(* Logix 5000 project; controller Sucrose_Main Emulate 5570 rev 20.12; software revision 20.01; part 4 of 30 *)
(* tags used below, declared in another part *)
   AI_E23_0 : REAL[8];   // Analog Input EN2T_FLX 192.168.1.23
   CIPRemote : Area_Program;
   SucroseCIP_PAUSED : BOOL;
   SucroseCIP_RECEIVING_LINE_REMOTE : CIP_REMOTE;
   SucroseCIP_RECEIVING_REMOTE : CIP_REMOTE;
   SucroseCIP_RINGMAIN_REMOTE : CIP_REMOTE;
   SucroseCIP_RUNNING : BOOL;
   SucroseCIP_SeatLift_Pulsing : BOOL;
   SucroseCIP_TK230101_REMOTE : CIP_REMOTE;
(* CIP_RemoteArea_AutoLogic, continued *)

ROUTINE CIP_Receiving_Line_Remote   (* ladder *)
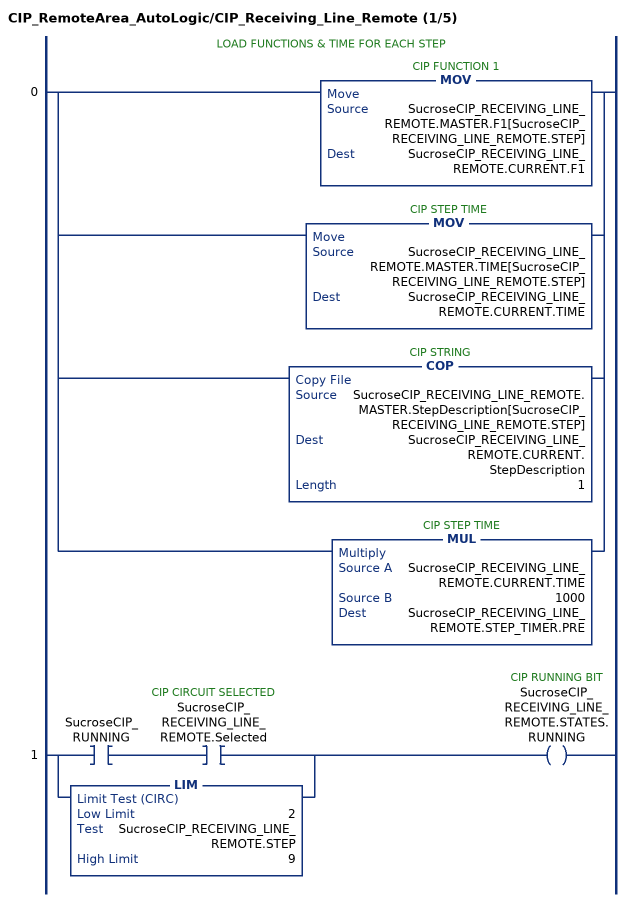
   // LOAD FUNCTIONS & TIME FOR EACH STEP
   0: [MOV(SucroseCIP_RECEIVING_LINE_REMOTE.MASTER.F1[SucroseCIP_RECEIVING_LINE_REMOTE.STEP],SucroseCIP_RECEIVING_LINE_REMOTE.CURRENT.F1) ,MOV(SucroseCIP_RECEIVING_LINE_REMOTE.MASTER.TIME[SucroseCIP_RECEIVING_LINE_REMOTE.STEP],SucroseCIP_RECEIVING_LINE_REMOTE.CURRENT.TIME) ,COP(SucroseCIP_RECEIVING_LINE_REMOTE.MASTER.StepDescription[SucroseCIP_RECEIVING_LINE_REMOTE.STEP],SucroseCIP_RECEIVING_LINE_REMOTE.CURRENT.StepDescription,1) ,MUL(SucroseCIP_RECEIVING_LINE_REMOTE.CURRENT.TIME,1000,SucroseCIP_RECEIVING_LINE_REMOTE.STEP_TIMER.PRE) ];
   1: [XIC(SucroseCIP_RUNNING) XIC(SucroseCIP_RECEIVING_LINE_REMOTE.Selected) ,LIM(2,SucroseCIP_RECEIVING_LINE_REMOTE.STEP,9) ]OTE(SucroseCIP_RECEIVING_LINE_REMOTE.STATES.RUNNING);
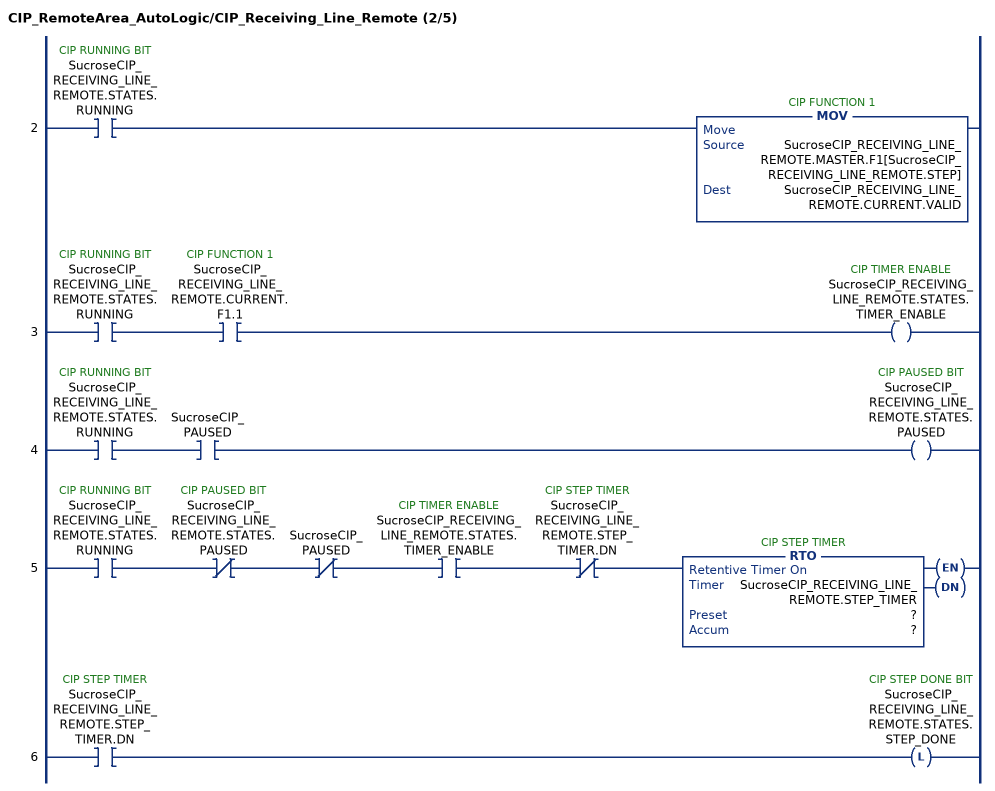
   2: XIC(SucroseCIP_RECEIVING_LINE_REMOTE.STATES.RUNNING)MOV(SucroseCIP_RECEIVING_LINE_REMOTE.MASTER.F1[SucroseCIP_RECEIVING_LINE_REMOTE.STEP],SucroseCIP_RECEIVING_LINE_REMOTE.CURRENT.VALID);
   3: XIC(SucroseCIP_RECEIVING_LINE_REMOTE.STATES.RUNNING)XIC(SucroseCIP_RECEIVING_LINE_REMOTE.CURRENT.F1.1)OTE(SucroseCIP_RECEIVING_LINE_REMOTE.STATES.TIMER_ENABLE);
   4: XIC(SucroseCIP_RECEIVING_LINE_REMOTE.STATES.RUNNING)XIC(SucroseCIP_PAUSED)OTE(SucroseCIP_RECEIVING_LINE_REMOTE.STATES.PAUSED);
   5: XIC(SucroseCIP_RECEIVING_LINE_REMOTE.STATES.RUNNING)XIO(SucroseCIP_RECEIVING_LINE_REMOTE.STATES.PAUSED)XIO(SucroseCIP_PAUSED)XIC(SucroseCIP_RECEIVING_LINE_REMOTE.STATES.TIMER_ENABLE)XIO(SucroseCIP_RECEIVING_LINE_REMOTE.STEP_TIMER.DN)RTO(SucroseCIP_RECEIVING_LINE_REMOTE.STEP_TIMER,?,?);
   6: XIC(SucroseCIP_RECEIVING_LINE_REMOTE.STEP_TIMER.DN)OTL(SucroseCIP_RECEIVING_LINE_REMOTE.STATES.STEP_DONE);
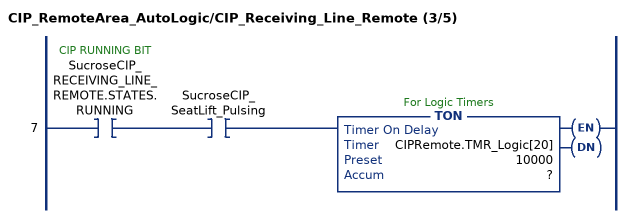
   7: XIC(SucroseCIP_RECEIVING_LINE_REMOTE.STATES.RUNNING)XIC(SucroseCIP_SeatLift_Pulsing)TON(CIPRemote.TMR_Logic[20],?,?);
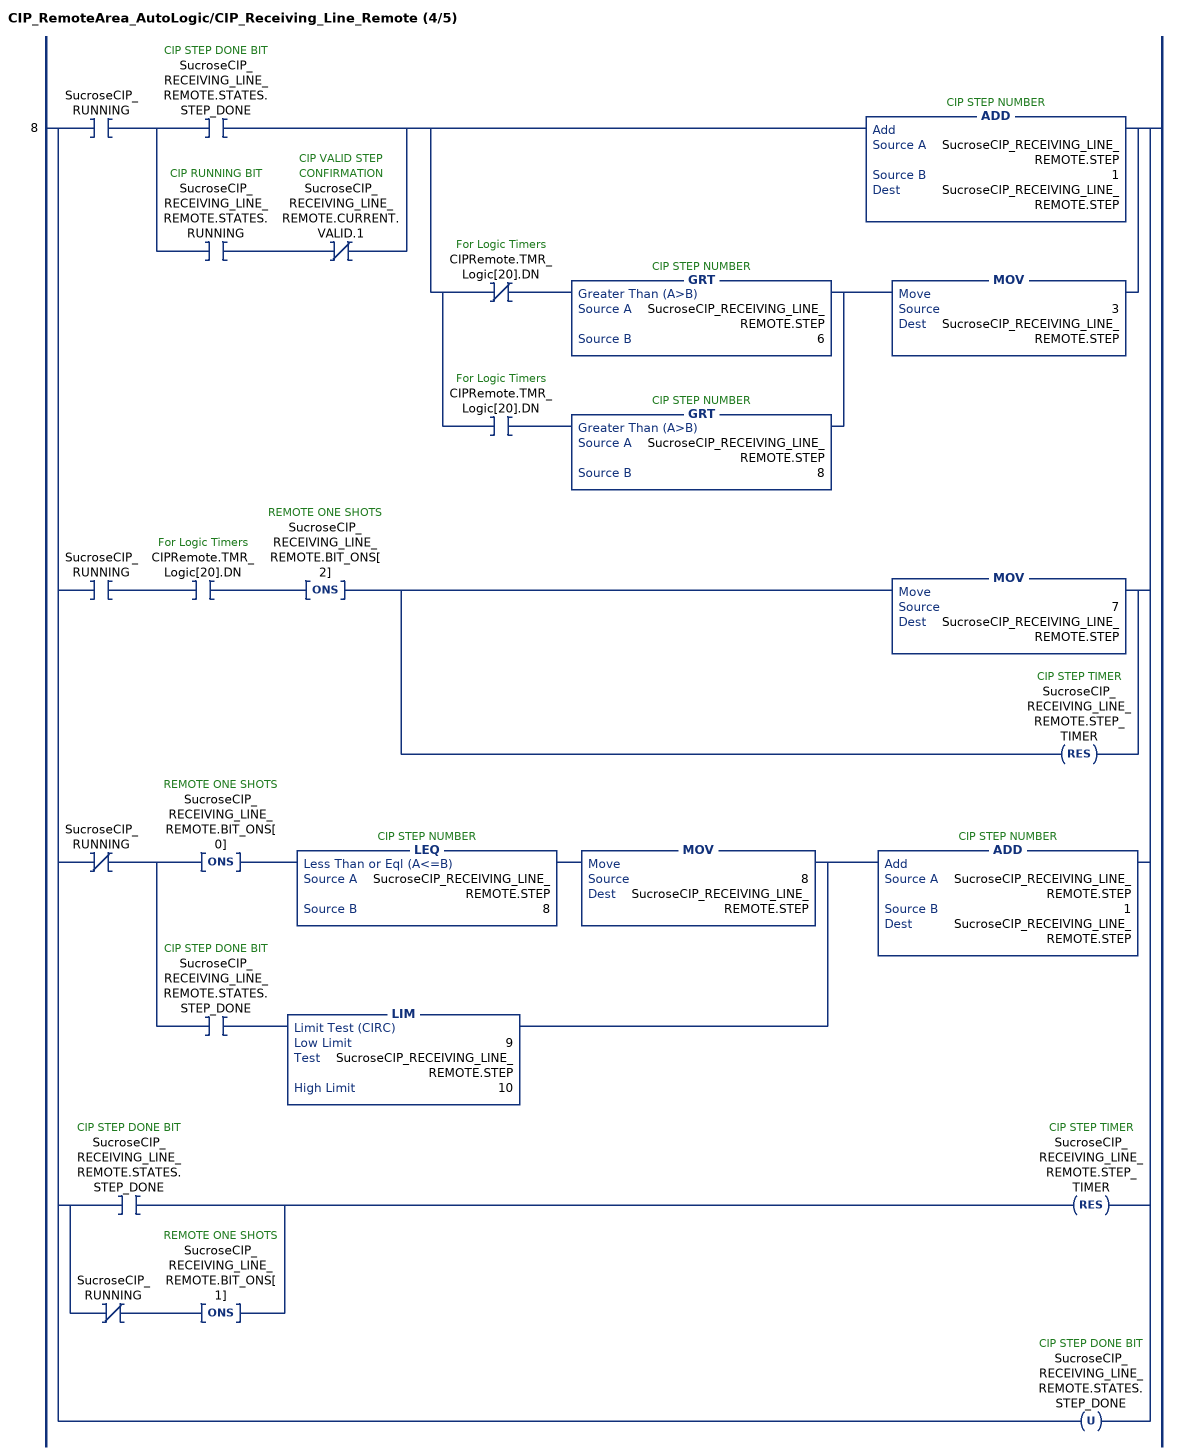
   8: [XIC(SucroseCIP_RUNNING) [XIC(SucroseCIP_RECEIVING_LINE_REMOTE.STATES.STEP_DONE) ,XIC(SucroseCIP_RECEIVING_LINE_REMOTE.STATES.RUNNING) XIO(SucroseCIP_RECEIVING_LINE_REMOTE.CURRENT.VALID.1) ] [ADD(SucroseCIP_RECEIVING_LINE_REMOTE.STEP,1,SucroseCIP_RECEIVING_LINE_REMOTE.STEP) ,[XIO(CIPRemote.TMR_Logic[20].DN) GRT(SucroseCIP_RECEIVING_LINE_REMOTE.STEP,6) ,XIC(CIPRemote.TMR_Logic[20].DN) GRT(SucroseCIP_RECEIVING_LINE_REMOTE.STEP,8) ] MOV(3,SucroseCIP_RECEIVING_LINE_REMOTE.STEP) ] ,XIC(SucroseCIP_RUNNING) XIC(CIPRemote.TMR_Logic[20].DN) ONS(SucroseCIP_RECEIVING_LINE_REMOTE.BIT_ONS[2]) [MOV(7,SucroseCIP_RECEIVING_LINE_REMOTE.STEP) ,RES(SucroseCIP_RECEIVING_LINE_REMOTE.STEP_TIMER) ] ,XIO(SucroseCIP_RUNNING) [ONS(SucroseCIP_RECEIVING_LINE_REMOTE.BIT_ONS[0]) LEQ(SucroseCIP_RECEIVING_LINE_REMOTE.STEP,8) MOV(8,SucroseCIP_RECEIVING_LINE_REMOTE.STEP) ,XIC(SucroseCIP_RECEIVING_LINE_REMOTE.STATES.STEP_DONE) LIM(9,SucroseCIP_RECEIVING_LINE_REMOTE.STEP,10) ] ADD(SucroseCIP_RECEIVING_LINE_REMOTE.STEP,1,SucroseCIP_RECEIVING_LINE_REMOTE.STEP) ,[XIC(SucroseCIP_RECEIVING_LINE_REMOTE.STATES.STEP_DONE) ,XIO(SucroseCIP_RUNNING) ONS(SucroseCIP_RECEIVING_LINE_REMOTE.BIT_ONS[1]) ] RES(SucroseCIP_RECEIVING_LINE_REMOTE.STEP_TIMER) ,OTU(SucroseCIP_RECEIVING_LINE_REMOTE.STATES.STEP_DONE) ];
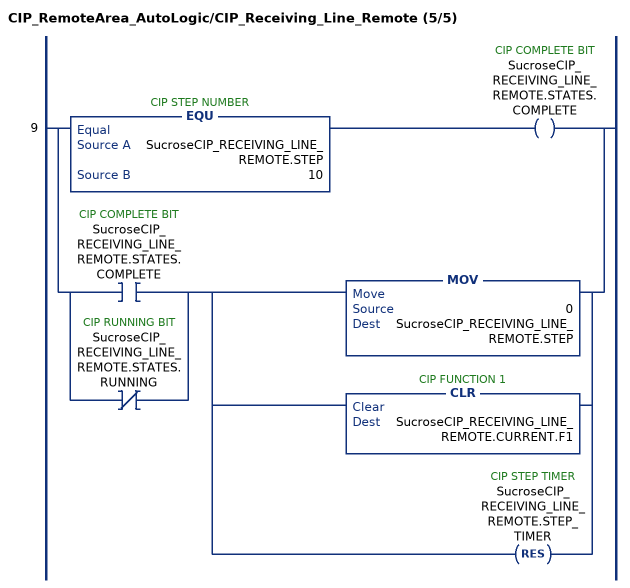
   9: [EQU(SucroseCIP_RECEIVING_LINE_REMOTE.STEP,10) OTE(SucroseCIP_RECEIVING_LINE_REMOTE.STATES.COMPLETE) ,[XIC(SucroseCIP_RECEIVING_LINE_REMOTE.STATES.COMPLETE) ,XIO(SucroseCIP_RECEIVING_LINE_REMOTE.STATES.RUNNING) ] [MOV(0,SucroseCIP_RECEIVING_LINE_REMOTE.STEP) ,CLR(SucroseCIP_RECEIVING_LINE_REMOTE.CURRENT.F1) ,RES(SucroseCIP_RECEIVING_LINE_REMOTE.STEP_TIMER) ] ];
END_ROUTINE

ROUTINE CIP_Receiving_Remote   (* ladder *)
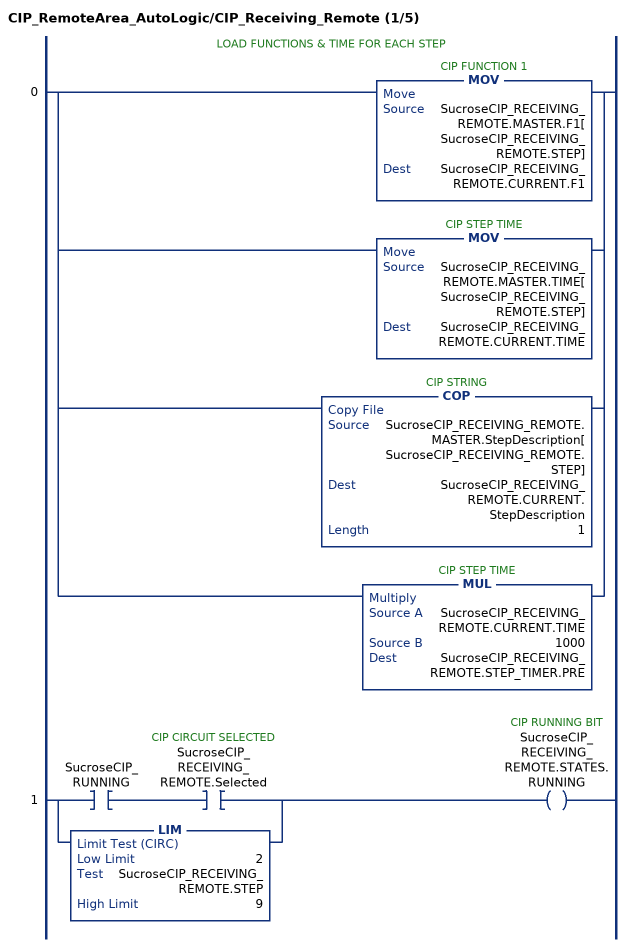
   // LOAD FUNCTIONS & TIME FOR EACH STEP
   0: [MOV(SucroseCIP_RECEIVING_REMOTE.MASTER.F1[SucroseCIP_RECEIVING_REMOTE.STEP],SucroseCIP_RECEIVING_REMOTE.CURRENT.F1) ,MOV(SucroseCIP_RECEIVING_REMOTE.MASTER.TIME[SucroseCIP_RECEIVING_REMOTE.STEP],SucroseCIP_RECEIVING_REMOTE.CURRENT.TIME) ,COP(SucroseCIP_RECEIVING_REMOTE.MASTER.StepDescription[SucroseCIP_RECEIVING_REMOTE.STEP],SucroseCIP_RECEIVING_REMOTE.CURRENT.StepDescription,1) ,MUL(SucroseCIP_RECEIVING_REMOTE.CURRENT.TIME,1000,SucroseCIP_RECEIVING_REMOTE.STEP_TIMER.PRE) ];
   1: [XIC(SucroseCIP_RUNNING) XIC(SucroseCIP_RECEIVING_REMOTE.Selected) ,LIM(2,SucroseCIP_RECEIVING_REMOTE.STEP,9) ]OTE(SucroseCIP_RECEIVING_REMOTE.STATES.RUNNING);
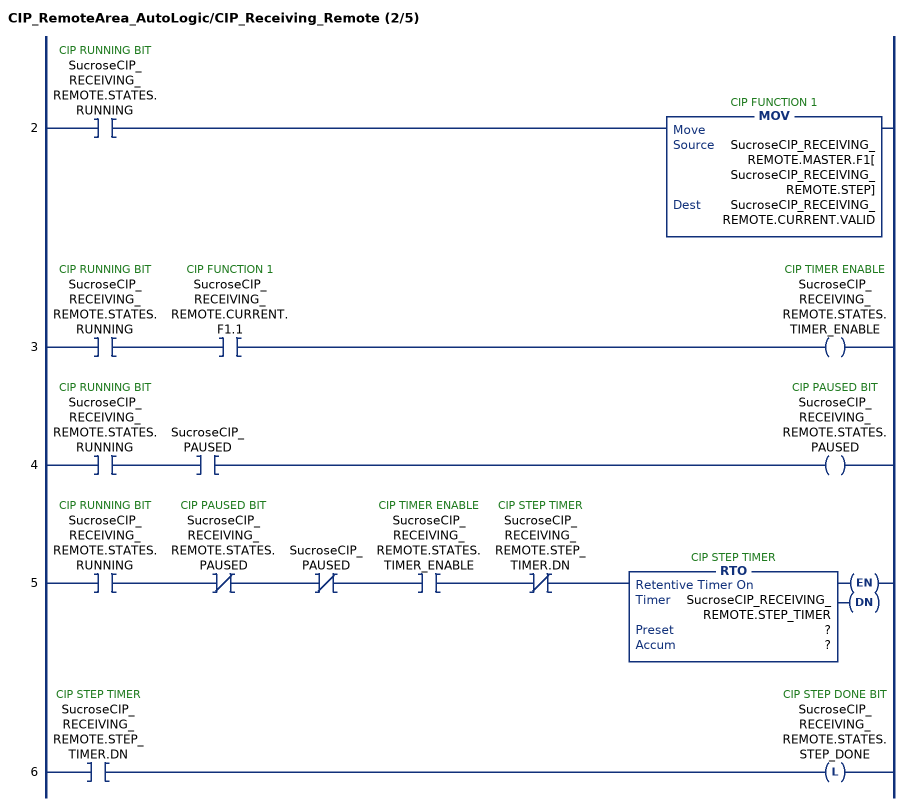
   2: XIC(SucroseCIP_RECEIVING_REMOTE.STATES.RUNNING)MOV(SucroseCIP_RECEIVING_REMOTE.MASTER.F1[SucroseCIP_RECEIVING_REMOTE.STEP],SucroseCIP_RECEIVING_REMOTE.CURRENT.VALID);
   3: XIC(SucroseCIP_RECEIVING_REMOTE.STATES.RUNNING)XIC(SucroseCIP_RECEIVING_REMOTE.CURRENT.F1.1)OTE(SucroseCIP_RECEIVING_REMOTE.STATES.TIMER_ENABLE);
   4: XIC(SucroseCIP_RECEIVING_REMOTE.STATES.RUNNING)XIC(SucroseCIP_PAUSED)OTE(SucroseCIP_RECEIVING_REMOTE.STATES.PAUSED);
   5: XIC(SucroseCIP_RECEIVING_REMOTE.STATES.RUNNING)XIO(SucroseCIP_RECEIVING_REMOTE.STATES.PAUSED)XIO(SucroseCIP_PAUSED)XIC(SucroseCIP_RECEIVING_REMOTE.STATES.TIMER_ENABLE)XIO(SucroseCIP_RECEIVING_REMOTE.STEP_TIMER.DN)RTO(SucroseCIP_RECEIVING_REMOTE.STEP_TIMER,?,?);
   6: XIC(SucroseCIP_RECEIVING_REMOTE.STEP_TIMER.DN)OTL(SucroseCIP_RECEIVING_REMOTE.STATES.STEP_DONE);
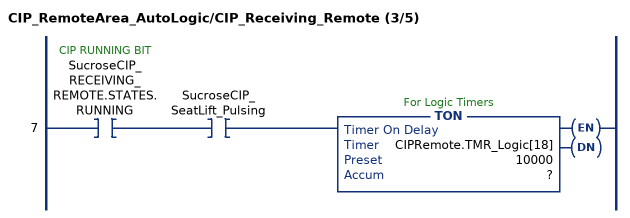
   7: XIC(SucroseCIP_RECEIVING_REMOTE.STATES.RUNNING)XIC(SucroseCIP_SeatLift_Pulsing)TON(CIPRemote.TMR_Logic[18],?,?);
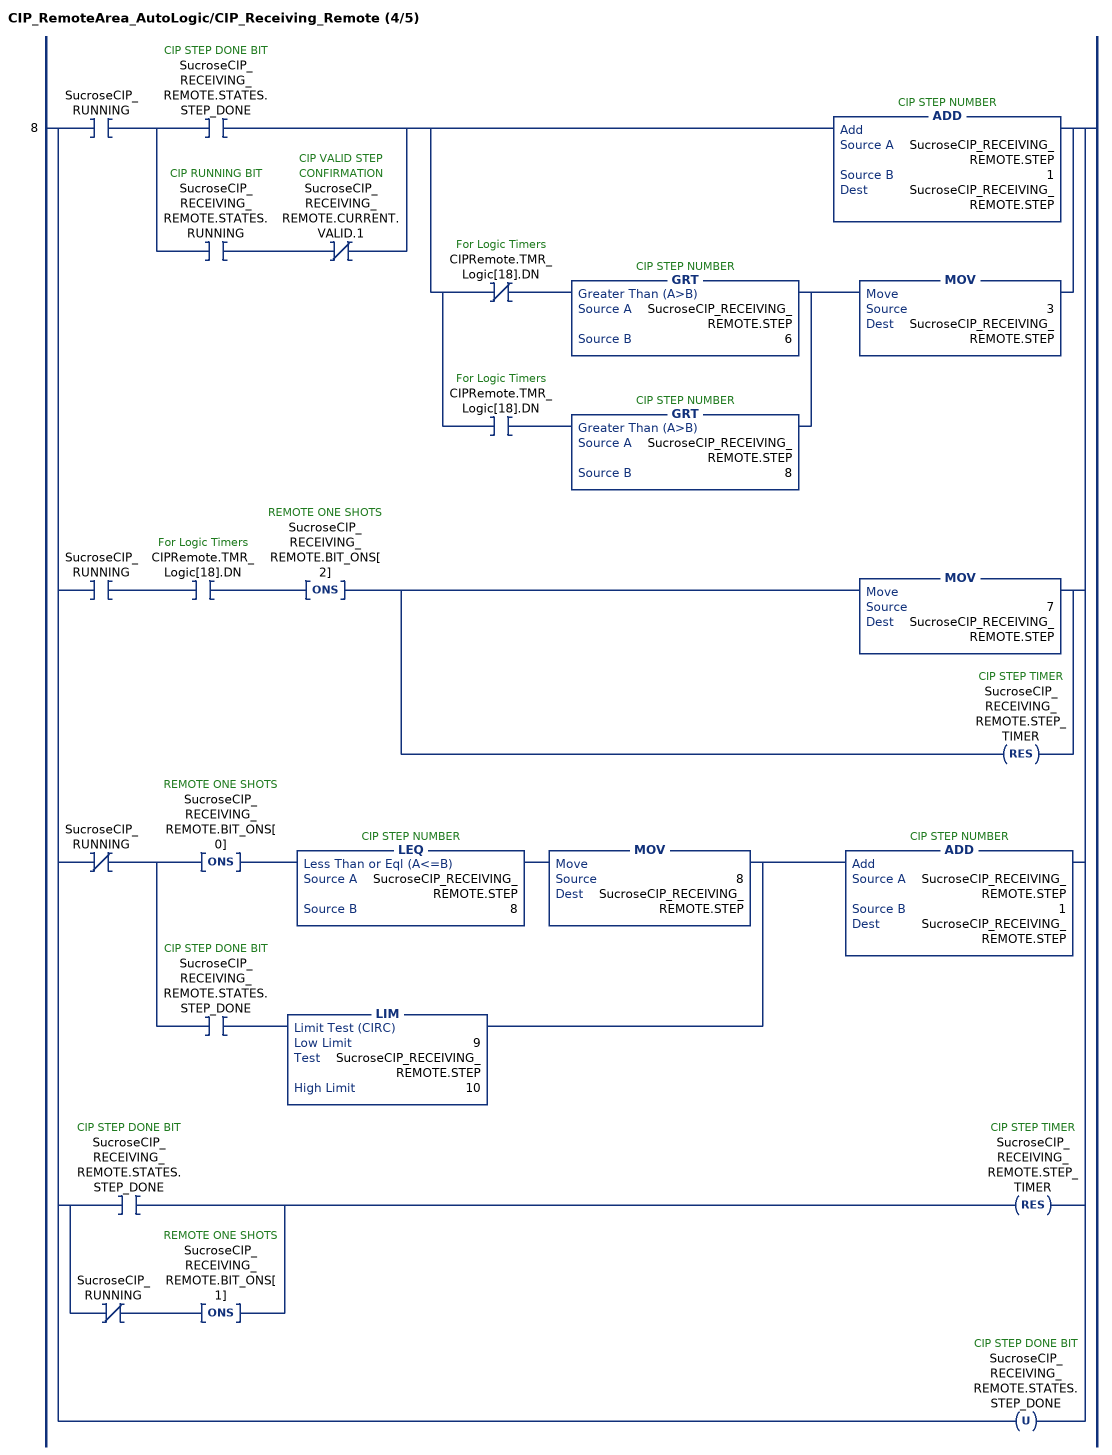
   8: [XIC(SucroseCIP_RUNNING) [XIC(SucroseCIP_RECEIVING_REMOTE.STATES.STEP_DONE) ,XIC(SucroseCIP_RECEIVING_REMOTE.STATES.RUNNING) XIO(SucroseCIP_RECEIVING_REMOTE.CURRENT.VALID.1) ] [ADD(SucroseCIP_RECEIVING_REMOTE.STEP,1,SucroseCIP_RECEIVING_REMOTE.STEP) ,[XIO(CIPRemote.TMR_Logic[18].DN) GRT(SucroseCIP_RECEIVING_REMOTE.STEP,6) ,XIC(CIPRemote.TMR_Logic[18].DN) GRT(SucroseCIP_RECEIVING_REMOTE.STEP,8) ] MOV(3,SucroseCIP_RECEIVING_REMOTE.STEP) ] ,XIC(SucroseCIP_RUNNING) XIC(CIPRemote.TMR_Logic[18].DN) ONS(SucroseCIP_RECEIVING_REMOTE.BIT_ONS[2]) [MOV(7,SucroseCIP_RECEIVING_REMOTE.STEP) ,RES(SucroseCIP_RECEIVING_REMOTE.STEP_TIMER) ] ,XIO(SucroseCIP_RUNNING) [ONS(SucroseCIP_RECEIVING_REMOTE.BIT_ONS[0]) LEQ(SucroseCIP_RECEIVING_REMOTE.STEP,8) MOV(8,SucroseCIP_RECEIVING_REMOTE.STEP) ,XIC(SucroseCIP_RECEIVING_REMOTE.STATES.STEP_DONE) LIM(9,SucroseCIP_RECEIVING_REMOTE.STEP,10) ] ADD(SucroseCIP_RECEIVING_REMOTE.STEP,1,SucroseCIP_RECEIVING_REMOTE.STEP) ,[XIC(SucroseCIP_RECEIVING_REMOTE.STATES.STEP_DONE) ,XIO(SucroseCIP_RUNNING) ONS(SucroseCIP_RECEIVING_REMOTE.BIT_ONS[1]) ] RES(SucroseCIP_RECEIVING_REMOTE.STEP_TIMER) ,OTU(SucroseCIP_RECEIVING_REMOTE.STATES.STEP_DONE) ];
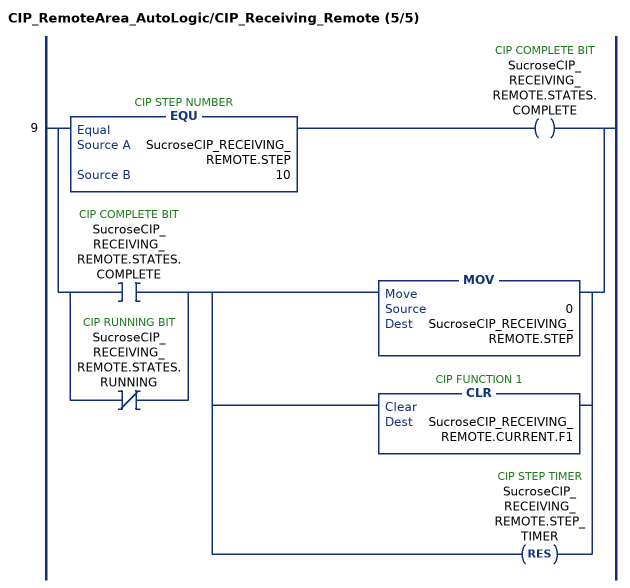
   9: [EQU(SucroseCIP_RECEIVING_REMOTE.STEP,10) OTE(SucroseCIP_RECEIVING_REMOTE.STATES.COMPLETE) ,[XIC(SucroseCIP_RECEIVING_REMOTE.STATES.COMPLETE) ,XIO(SucroseCIP_RECEIVING_REMOTE.STATES.RUNNING) ] [MOV(0,SucroseCIP_RECEIVING_REMOTE.STEP) ,CLR(SucroseCIP_RECEIVING_REMOTE.CURRENT.F1) ,RES(SucroseCIP_RECEIVING_REMOTE.STEP_TIMER) ] ];
END_ROUTINE

ROUTINE CIP_RingMain_Remote   (* ladder *)
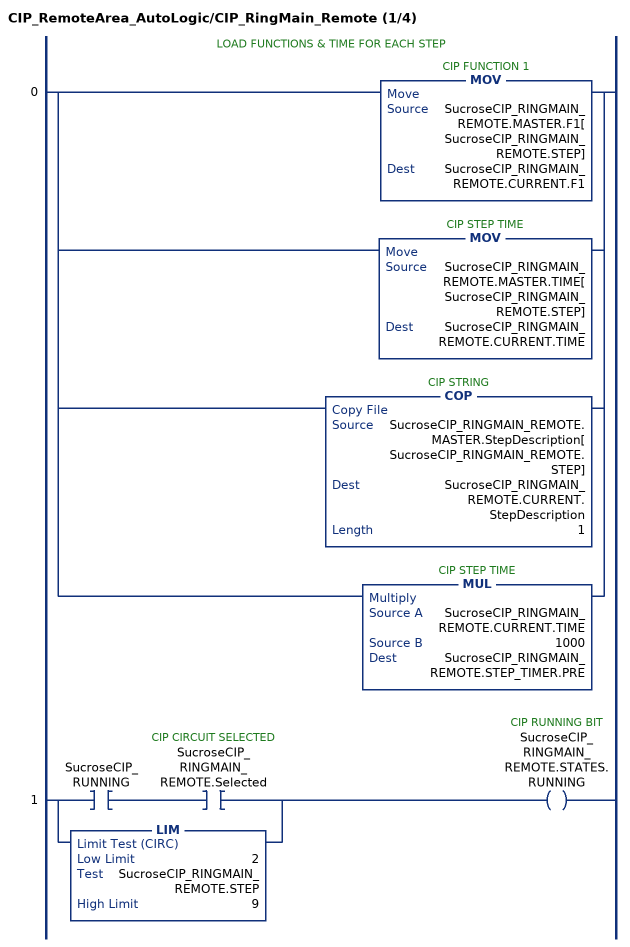
   // LOAD FUNCTIONS & TIME FOR EACH STEP
   0: [MOV(SucroseCIP_RINGMAIN_REMOTE.MASTER.F1[SucroseCIP_RINGMAIN_REMOTE.STEP],SucroseCIP_RINGMAIN_REMOTE.CURRENT.F1) ,MOV(SucroseCIP_RINGMAIN_REMOTE.MASTER.TIME[SucroseCIP_RINGMAIN_REMOTE.STEP],SucroseCIP_RINGMAIN_REMOTE.CURRENT.TIME) ,COP(SucroseCIP_RINGMAIN_REMOTE.MASTER.StepDescription[SucroseCIP_RINGMAIN_REMOTE.STEP],SucroseCIP_RINGMAIN_REMOTE.CURRENT.StepDescription,1) ,MUL(SucroseCIP_RINGMAIN_REMOTE.CURRENT.TIME,1000,SucroseCIP_RINGMAIN_REMOTE.STEP_TIMER.PRE) ];
   1: [XIC(SucroseCIP_RUNNING) XIC(SucroseCIP_RINGMAIN_REMOTE.Selected) ,LIM(2,SucroseCIP_RINGMAIN_REMOTE.STEP,9) ]OTE(SucroseCIP_RINGMAIN_REMOTE.STATES.RUNNING);
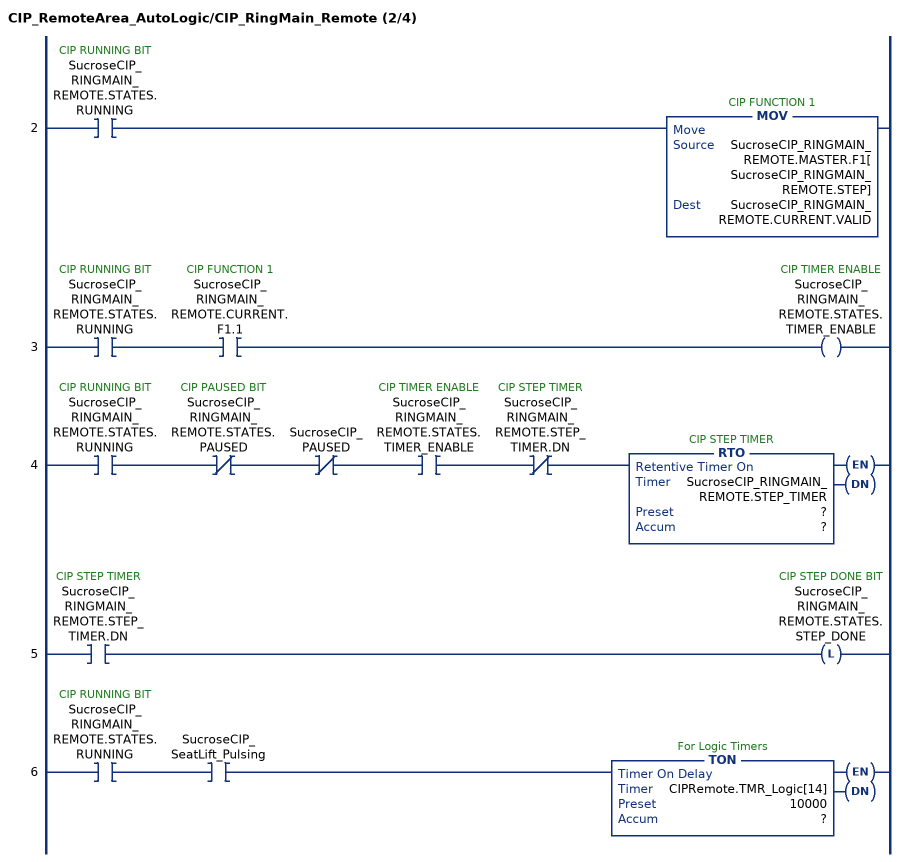
   2: XIC(SucroseCIP_RINGMAIN_REMOTE.STATES.RUNNING)MOV(SucroseCIP_RINGMAIN_REMOTE.MASTER.F1[SucroseCIP_RINGMAIN_REMOTE.STEP],SucroseCIP_RINGMAIN_REMOTE.CURRENT.VALID);
   3: XIC(SucroseCIP_RINGMAIN_REMOTE.STATES.RUNNING)XIC(SucroseCIP_RINGMAIN_REMOTE.CURRENT.F1.1)OTE(SucroseCIP_RINGMAIN_REMOTE.STATES.TIMER_ENABLE);
   4: XIC(SucroseCIP_RINGMAIN_REMOTE.STATES.RUNNING)XIO(SucroseCIP_RINGMAIN_REMOTE.STATES.PAUSED)XIO(SucroseCIP_PAUSED)XIC(SucroseCIP_RINGMAIN_REMOTE.STATES.TIMER_ENABLE)XIO(SucroseCIP_RINGMAIN_REMOTE.STEP_TIMER.DN)RTO(SucroseCIP_RINGMAIN_REMOTE.STEP_TIMER,?,?);
   5: XIC(SucroseCIP_RINGMAIN_REMOTE.STEP_TIMER.DN)OTL(SucroseCIP_RINGMAIN_REMOTE.STATES.STEP_DONE);
   6: XIC(SucroseCIP_RINGMAIN_REMOTE.STATES.RUNNING)XIC(SucroseCIP_SeatLift_Pulsing)TON(CIPRemote.TMR_Logic[14],?,?);
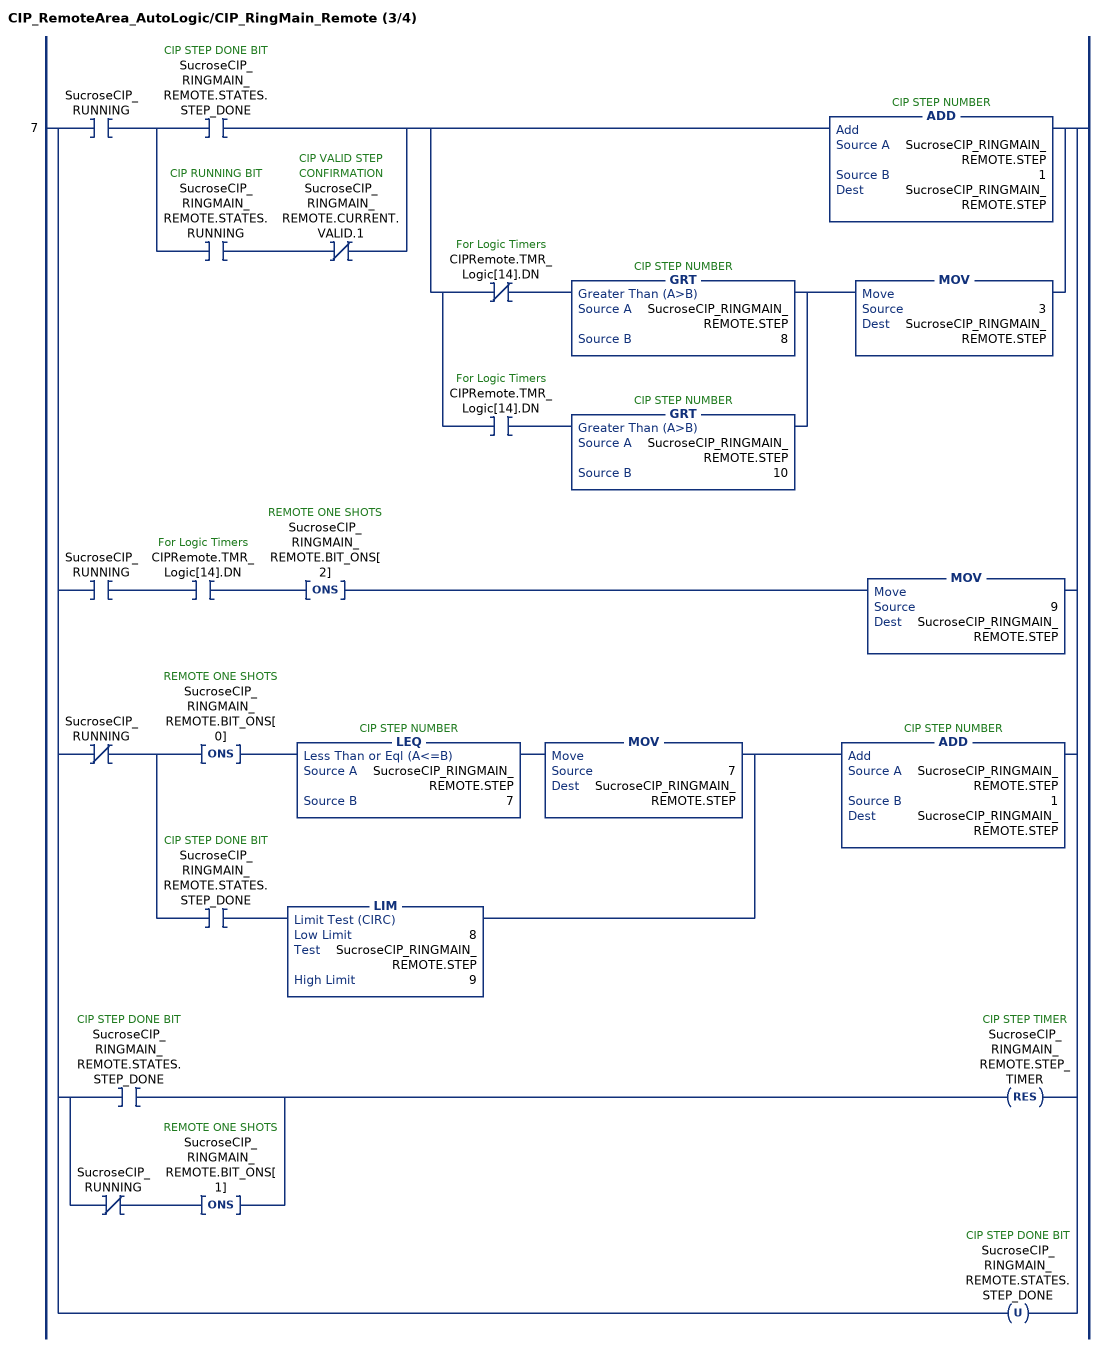
   7: [XIC(SucroseCIP_RUNNING) [XIC(SucroseCIP_RINGMAIN_REMOTE.STATES.STEP_DONE) ,XIC(SucroseCIP_RINGMAIN_REMOTE.STATES.RUNNING) XIO(SucroseCIP_RINGMAIN_REMOTE.CURRENT.VALID.1) ] [ADD(SucroseCIP_RINGMAIN_REMOTE.STEP,1,SucroseCIP_RINGMAIN_REMOTE.STEP) ,[XIO(CIPRemote.TMR_Logic[14].DN) GRT(SucroseCIP_RINGMAIN_REMOTE.STEP,8) ,XIC(CIPRemote.TMR_Logic[14].DN) GRT(SucroseCIP_RINGMAIN_REMOTE.STEP,10) ] MOV(3,SucroseCIP_RINGMAIN_REMOTE.STEP) ] ,XIC(SucroseCIP_RUNNING) XIC(CIPRemote.TMR_Logic[14].DN) ONS(SucroseCIP_RINGMAIN_REMOTE.BIT_ONS[2]) MOV(9,SucroseCIP_RINGMAIN_REMOTE.STEP) ,XIO(SucroseCIP_RUNNING) [ONS(SucroseCIP_RINGMAIN_REMOTE.BIT_ONS[0]) LEQ(SucroseCIP_RINGMAIN_REMOTE.STEP,7) MOV(7,SucroseCIP_RINGMAIN_REMOTE.STEP) ,XIC(SucroseCIP_RINGMAIN_REMOTE.STATES.STEP_DONE) LIM(8,SucroseCIP_RINGMAIN_REMOTE.STEP,9) ] ADD(SucroseCIP_RINGMAIN_REMOTE.STEP,1,SucroseCIP_RINGMAIN_REMOTE.STEP) ,[XIC(SucroseCIP_RINGMAIN_REMOTE.STATES.STEP_DONE) ,XIO(SucroseCIP_RUNNING) ONS(SucroseCIP_RINGMAIN_REMOTE.BIT_ONS[1]) ] RES(SucroseCIP_RINGMAIN_REMOTE.STEP_TIMER) ,OTU(SucroseCIP_RINGMAIN_REMOTE.STATES.STEP_DONE) ];
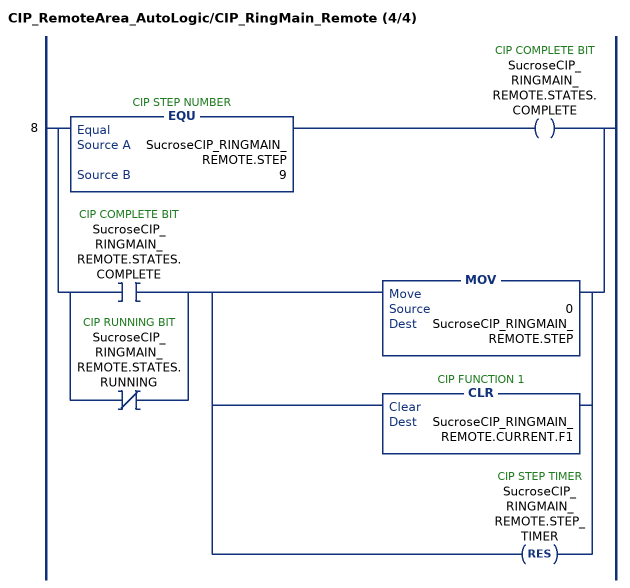
   8: [EQU(SucroseCIP_RINGMAIN_REMOTE.STEP,9) OTE(SucroseCIP_RINGMAIN_REMOTE.STATES.COMPLETE) ,[XIC(SucroseCIP_RINGMAIN_REMOTE.STATES.COMPLETE) ,XIO(SucroseCIP_RINGMAIN_REMOTE.STATES.RUNNING) ] [MOV(0,SucroseCIP_RINGMAIN_REMOTE.STEP) ,CLR(SucroseCIP_RINGMAIN_REMOTE.CURRENT.F1) ,RES(SucroseCIP_RINGMAIN_REMOTE.STEP_TIMER) ] ];
END_ROUTINE

ROUTINE CIP_TK230101_Remote   (* ladder *)
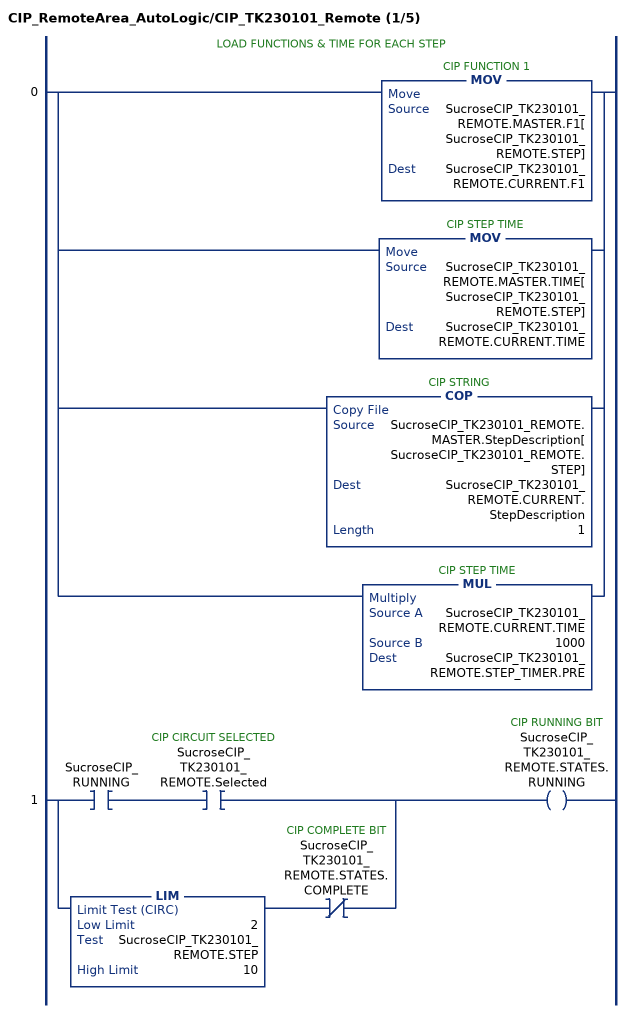
   // LOAD FUNCTIONS & TIME FOR EACH STEP
   0: [MOV(SucroseCIP_TK230101_REMOTE.MASTER.F1[SucroseCIP_TK230101_REMOTE.STEP],SucroseCIP_TK230101_REMOTE.CURRENT.F1) ,MOV(SucroseCIP_TK230101_REMOTE.MASTER.TIME[SucroseCIP_TK230101_REMOTE.STEP],SucroseCIP_TK230101_REMOTE.CURRENT.TIME) ,COP(SucroseCIP_TK230101_REMOTE.MASTER.StepDescription[SucroseCIP_TK230101_REMOTE.STEP],SucroseCIP_TK230101_REMOTE.CURRENT.StepDescription,1) ,MUL(SucroseCIP_TK230101_REMOTE.CURRENT.TIME,1000,SucroseCIP_TK230101_REMOTE.STEP_TIMER.PRE) ];
   1: [XIC(SucroseCIP_RUNNING) XIC(SucroseCIP_TK230101_REMOTE.Selected) ,LIM(2,SucroseCIP_TK230101_REMOTE.STEP,10) XIO(SucroseCIP_TK230101_REMOTE.STATES.COMPLETE) ]OTE(SucroseCIP_TK230101_REMOTE.STATES.RUNNING);
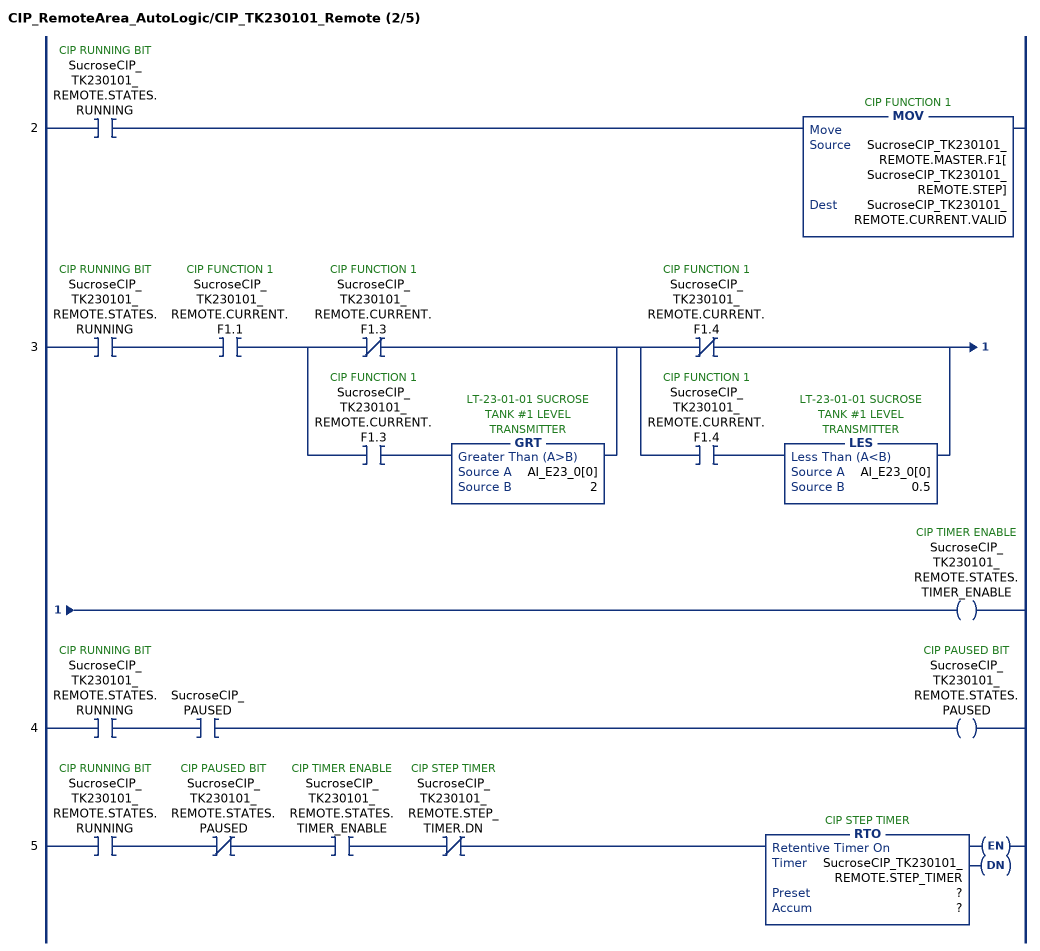
   2: XIC(SucroseCIP_TK230101_REMOTE.STATES.RUNNING)MOV(SucroseCIP_TK230101_REMOTE.MASTER.F1[SucroseCIP_TK230101_REMOTE.STEP],SucroseCIP_TK230101_REMOTE.CURRENT.VALID);
   3: XIC(SucroseCIP_TK230101_REMOTE.STATES.RUNNING)XIC(SucroseCIP_TK230101_REMOTE.CURRENT.F1.1)[XIO(SucroseCIP_TK230101_REMOTE.CURRENT.F1.3) ,XIC(SucroseCIP_TK230101_REMOTE.CURRENT.F1.3) GRT(AI_E23_0[0],2) ][XIO(SucroseCIP_TK230101_REMOTE.CURRENT.F1.4) ,XIC(SucroseCIP_TK230101_REMOTE.CURRENT.F1.4) LES(AI_E23_0[0],0.5) ]OTE(SucroseCIP_TK230101_REMOTE.STATES.TIMER_ENABLE);
   4: XIC(SucroseCIP_TK230101_REMOTE.STATES.RUNNING)XIC(SucroseCIP_PAUSED)OTE(SucroseCIP_TK230101_REMOTE.STATES.PAUSED);
   5: XIC(SucroseCIP_TK230101_REMOTE.STATES.RUNNING)XIO(SucroseCIP_TK230101_REMOTE.STATES.PAUSED)XIC(SucroseCIP_TK230101_REMOTE.STATES.TIMER_ENABLE)XIO(SucroseCIP_TK230101_REMOTE.STEP_TIMER.DN)RTO(SucroseCIP_TK230101_REMOTE.STEP_TIMER,?,?);
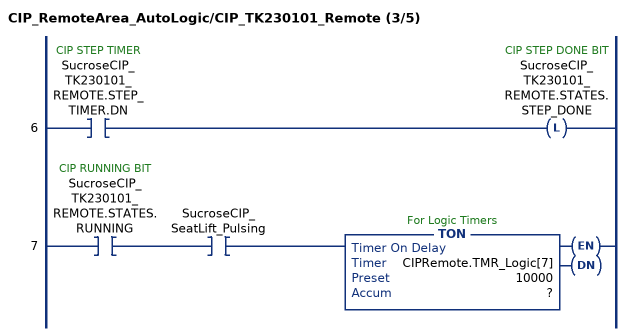
   6: XIC(SucroseCIP_TK230101_REMOTE.STEP_TIMER.DN)OTL(SucroseCIP_TK230101_REMOTE.STATES.STEP_DONE);
   7: XIC(SucroseCIP_TK230101_REMOTE.STATES.RUNNING)XIC(SucroseCIP_SeatLift_Pulsing)TON(CIPRemote.TMR_Logic[7],?,?);
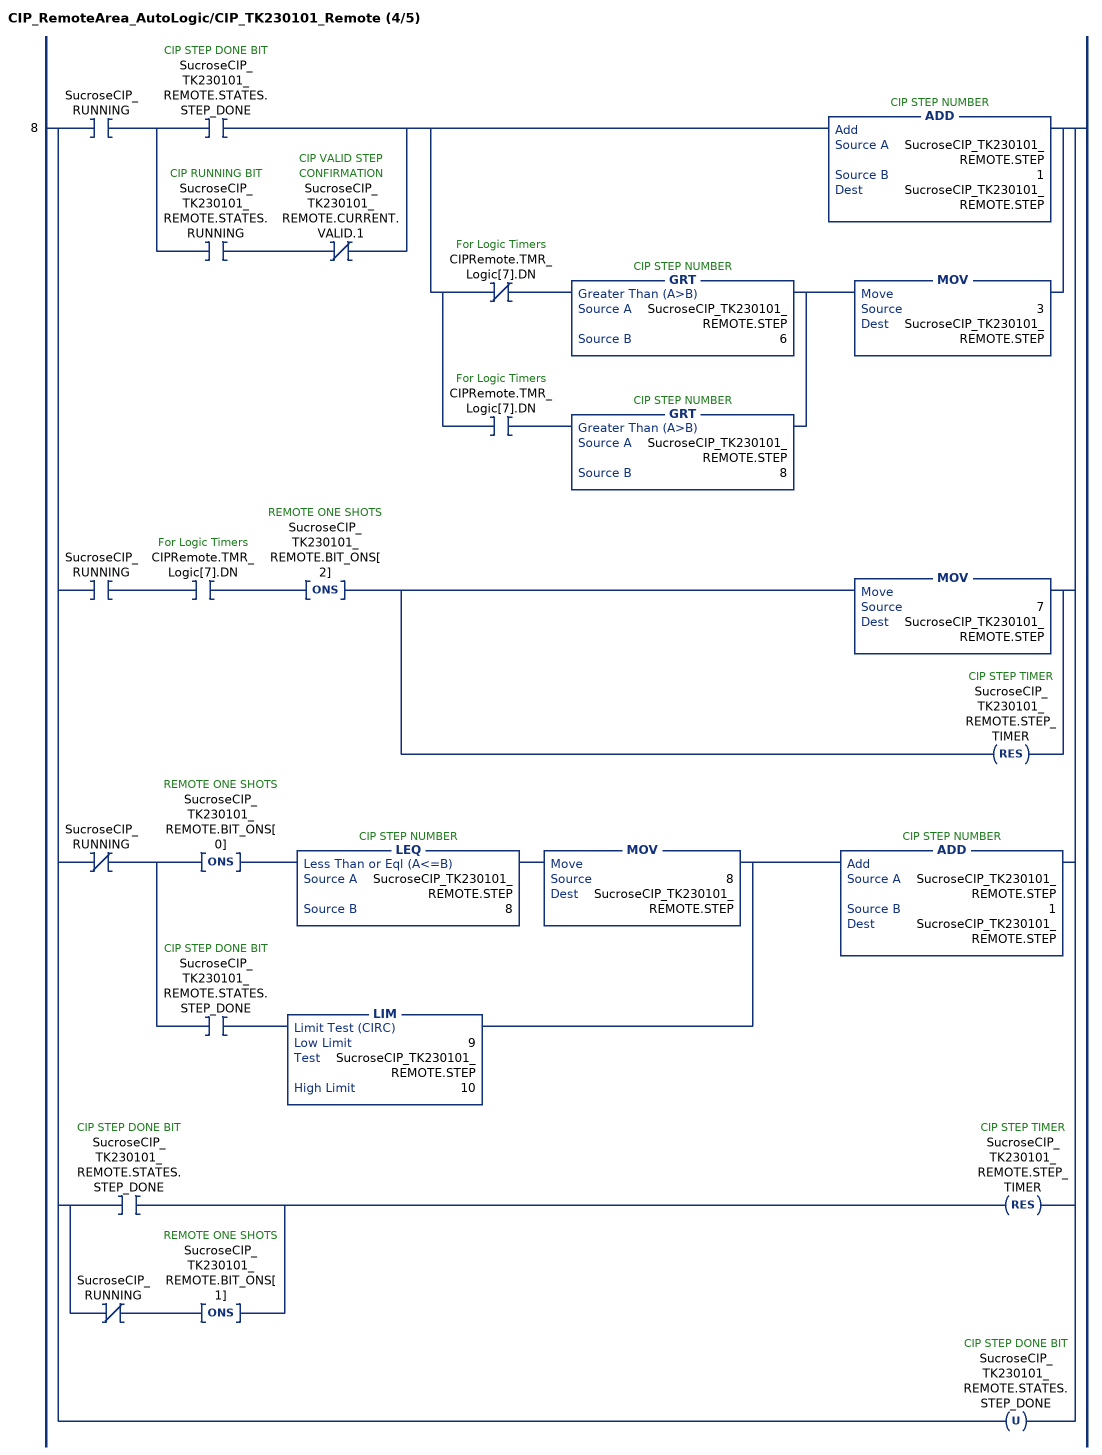
   8: [XIC(SucroseCIP_RUNNING) [XIC(SucroseCIP_TK230101_REMOTE.STATES.STEP_DONE) ,XIC(SucroseCIP_TK230101_REMOTE.STATES.RUNNING) XIO(SucroseCIP_TK230101_REMOTE.CURRENT.VALID.1) ] [ADD(SucroseCIP_TK230101_REMOTE.STEP,1,SucroseCIP_TK230101_REMOTE.STEP) ,[XIO(CIPRemote.TMR_Logic[7].DN) GRT(SucroseCIP_TK230101_REMOTE.STEP,6) ,XIC(CIPRemote.TMR_Logic[7].DN) GRT(SucroseCIP_TK230101_REMOTE.STEP,8) ] MOV(3,SucroseCIP_TK230101_REMOTE.STEP) ] ,XIC(SucroseCIP_RUNNING) XIC(CIPRemote.TMR_Logic[7].DN) ONS(SucroseCIP_TK230101_REMOTE.BIT_ONS[2]) [MOV(7,SucroseCIP_TK230101_REMOTE.STEP) ,RES(SucroseCIP_TK230101_REMOTE.STEP_TIMER) ] ,XIO(SucroseCIP_RUNNING) [ONS(SucroseCIP_TK230101_REMOTE.BIT_ONS[0]) LEQ(SucroseCIP_TK230101_REMOTE.STEP,8) MOV(8,SucroseCIP_TK230101_REMOTE.STEP) ,XIC(SucroseCIP_TK230101_REMOTE.STATES.STEP_DONE) LIM(9,SucroseCIP_TK230101_REMOTE.STEP,10) ] ADD(SucroseCIP_TK230101_REMOTE.STEP,1,SucroseCIP_TK230101_REMOTE.STEP) ,[XIC(SucroseCIP_TK230101_REMOTE.STATES.STEP_DONE) ,XIO(SucroseCIP_RUNNING) ONS(SucroseCIP_TK230101_REMOTE.BIT_ONS[1]) ] RES(SucroseCIP_TK230101_REMOTE.STEP_TIMER) ,OTU(SucroseCIP_TK230101_REMOTE.STATES.STEP_DONE) ];
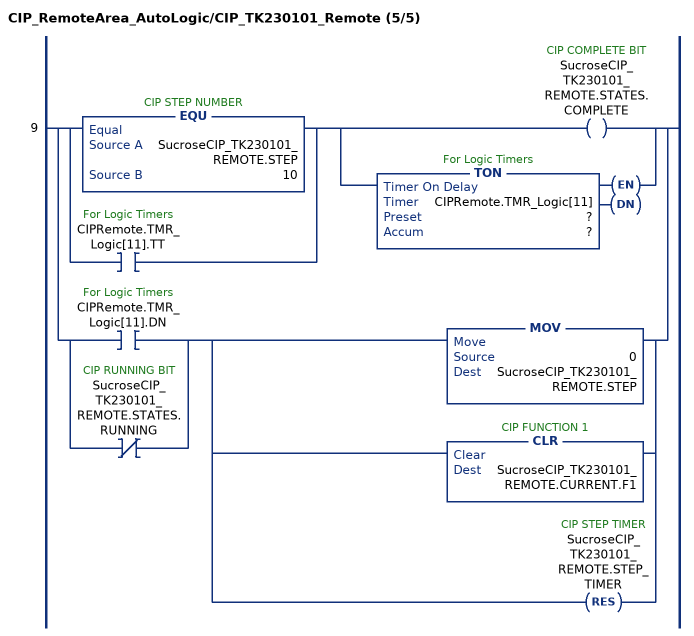
   9: [[EQU(SucroseCIP_TK230101_REMOTE.STEP,10) ,XIC(CIPRemote.TMR_Logic[11].TT) ] [OTE(SucroseCIP_TK230101_REMOTE.STATES.COMPLETE) ,TON(CIPRemote.TMR_Logic[11],?,?) ] ,[XIC(CIPRemote.TMR_Logic[11].DN) ,XIO(SucroseCIP_TK230101_REMOTE.STATES.RUNNING) ] [MOV(0,SucroseCIP_TK230101_REMOTE.STEP) ,CLR(SucroseCIP_TK230101_REMOTE.CURRENT.F1) ,RES(SucroseCIP_TK230101_REMOTE.STEP_TIMER) ] ];
END_ROUTINE
